# EPICS autosave request: ampMotorApp/Db/STAC5_positions.req
#
# STAC5 Motor Settings
#
# Author: Wesley Moore (wmoore@jlab.org)
# Date:   Oct 2013
#
# !!! DO NOT RESTORE - FOR REFERENCE ONLY !!!
$(P)$(R)POS
